(* IEC 61131-3 sources: st-fmt/tests/fixtures/declarations, 10 files *)

(* ---- types.expected.st ---- *)
VAR_GLOBAL
    a : INT;
    b : ARRAY [0..9] OF INT;
    c : ARRAY [0..3, 1..2] OF REAL;
    d : ARRAY [0..MAX_DEVICES - 1] OF BOOL;
    e : STRING[512];
    f : STRING(80);
    g : POINTER TO INT;
    h : REFERENCE TO MyStruct;
    i : CmpApp.EVTPARAM_CmpApp;
    j : ARRAY [0..1] OF ARRAY [0..2] OF INT;
    k : POINTER TO ARRAY [0..2] OF INT;
END_VAR

(* ---- types.st ---- *)
VAR_GLOBAL
a : int;
b : ARRAY[0..9] OF int;
c : ARRAY [0..3, 1..2] OF real;
d : ARRAY [0..MAX_DEVICES - 1] OF bool;
e : STRING [512];
f : STRING(80);
g : pointer to int;
h : reference to MyStruct;
i : CmpApp.EVTPARAM_CmpApp;
j : ARRAY [0..1] OF ARRAY [0..2] OF INT;
k : pointer to ARRAY [0..2] OF int;
END_VAR

(* ---- var_alignment.expected.st ---- *)
VAR_GLOBAL
    bEnable       : BOOL := FALSE;
    // grouping note
    nCount        : INT;
    rVeryLongName : REAL := 20.5;

    sShort : STRING[80];
END_VAR

(* ---- var_alignment.st ---- *)
VAR_GLOBAL
bEnable : BOOL := FALSE;
// grouping note
nCount:INT;
rVeryLongName:REAL:=20.5;

sShort : STRING[80];
END_VAR

(* ---- var_initializers.expected.st ---- *)
VAR_GLOBAL
    aSmall  : ARRAY [0..2] OF INT  := [1, 2, 3];
    aRepeat : ARRAY [0..9] OF INT  := [10(0)];
    aBig    : ARRAY [0..19] OF INT := [
        1000, 2000, 3000, 4000, 5000, 6000, 7000, 8000, 9000, 10000, 11000, 12000, 13000, 14000
    ];
    stPoint : Point                := (x := 1, y := 2);
    stWide  : Config               := (
        nFirstSetting  := 1,
        nSecondSetting := 2,
        nThirdSetting  := 3,
        nFourth        := 4,
    );
    sText   : STRING[80]           := 'hello';
END_VAR

(* ---- var_initializers.st ---- *)
VAR_GLOBAL
aSmall : ARRAY [0..2] OF INT := [1,2,3];
aRepeat : ARRAY [0..9] OF INT := [10(0)];
aBig : ARRAY [0..19] OF INT := [1000,2000,3000,4000,5000,6000,7000,8000,9000,10000,11000,12000,13000,14000];
stPoint : Point := (x := 1, y := 2);
stWide : Config := (nFirstSetting := 1, nSecondSetting := 2, nThirdSetting := 3, nFourth := 4);
sText : STRING[80] := 'hello';
END_VAR

(* ---- var_locations.expected.st ---- *)
VAR_GLOBAL
    bStart AT %IX0.0 : BOOL;
    bStop  AT %IX0.1 : BOOL;
    nCount           : INT;
END_VAR

(* ---- var_locations.st ---- *)
VAR_GLOBAL
bStart AT %ix0.0 : BOOL;
bStop at %IX0.1:BOOL;
nCount : INT;
END_VAR

(* ---- var_qualifiers.expected.st ---- *)
VAR_GLOBAL CONSTANT
    MAX_ITEMS : INT := 100;
END_VAR

VAR_GLOBAL RETAIN PERSISTENT
    nCycles : UDINT;
END_VAR

(* ---- var_qualifiers.st ---- *)
var_global constant
MAX_ITEMS : int := 100;
end_var
VAR_GLOBAL retain persistent
nCycles : udint;
END_VAR
